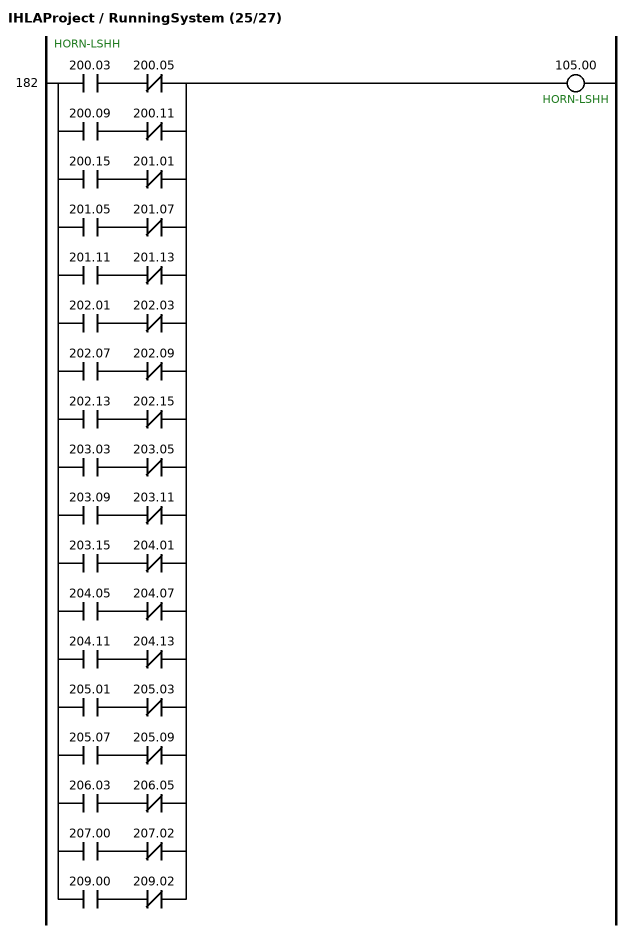
; [picture p24: IHLAProject / RunningSystem, rungs 182-182]
; rung 182: HORN-LSHH
LD 200.03
ANDNOT 200.05
LD 200.09
ANDNOT 200.11
ORLD
LD 200.15
ANDNOT 201.01
ORLD
LD 201.05
ANDNOT 201.07
ORLD
LD 201.11
ANDNOT 201.13
ORLD
LD 202.01
ANDNOT 202.03
ORLD
LD 202.07
ANDNOT 202.09
ORLD
LD 202.13
ANDNOT 202.15
ORLD
LD 203.03
ANDNOT 203.05
ORLD
LD 203.09
ANDNOT 203.11
ORLD
LD 203.15
ANDNOT 204.01
ORLD
LD 204.05
ANDNOT 204.07
ORLD
LD 204.11
ANDNOT 204.13
ORLD
LD 205.01
ANDNOT 205.03
ORLD
LD 205.07
ANDNOT 205.09
ORLD
LD 206.03
ANDNOT 206.05
ORLD
LD 207.00
ANDNOT 207.02
ORLD
LD 209.00
ANDNOT 209.02
ORLD
OUT 105.00  ; HORN-LSHH

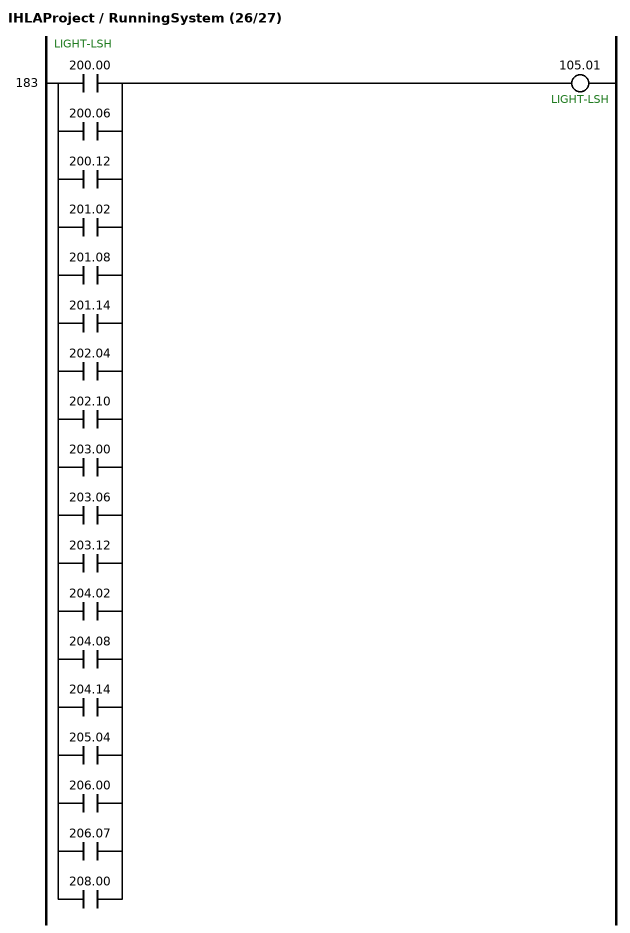
; rung 183: LIGHT-LSH
LD 200.00
OR 200.06
OR 200.12
OR 201.02
OR 201.08
OR 201.14
OR 202.04
OR 202.10
OR 203.00
OR 203.06
OR 203.12
OR 204.02
OR 204.08
OR 204.14
OR 205.04
OR 206.00
OR 206.07
OR 208.00
OUT 105.01  ; LIGHT-LSH

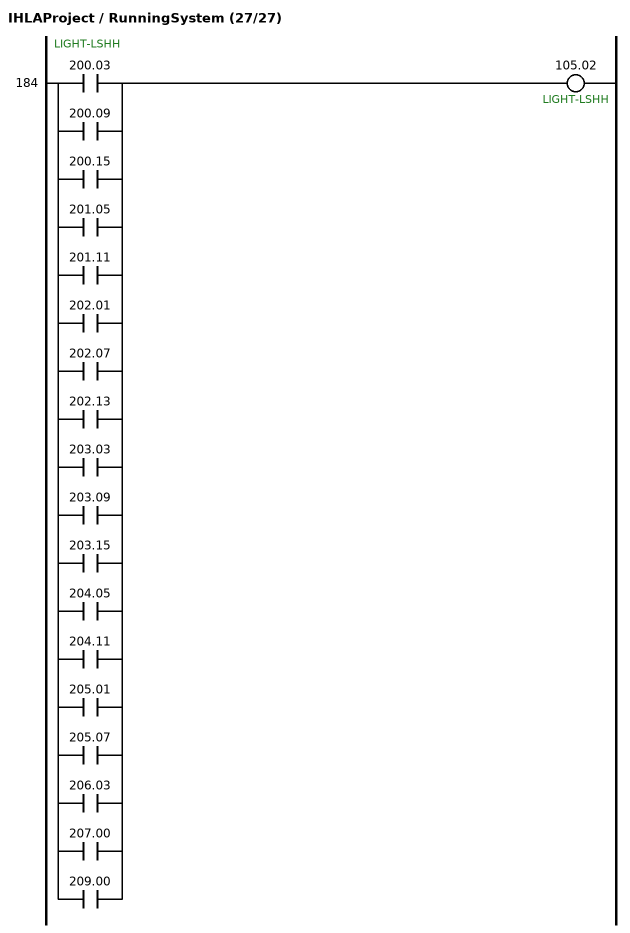
; rung 184: LIGHT-LSHH
LD 200.03
OR 200.09
OR 200.15
OR 201.05
OR 201.11
OR 202.01
OR 202.07
OR 202.13
OR 203.03
OR 203.09
OR 203.15
OR 204.05
OR 204.11
OR 205.01
OR 205.07
OR 206.03
OR 207.00
OR 209.00
OUT 105.02  ; LIGHT-LSHH

### Section END
; rung 0
END(001)